// TIA Portal project "Esteira_seletora" (V17)

(* hardware
DEVICE "S7-1500/ET200MP station_1"  S7-1500 station
   slot 0: "Rail_0"  Rack  6ES7 590-1***0-0AA0
   slot 1: "PLC_1"  CPU 1516-3 PN/DP  6ES7 516-3AN02-0AB0  V2.9
      slot 3: "CPU display_1"  6ES7591-1BA00-0AA0
      slot 32768: "PROFINET interface_1"  X1
      slot 33024: "PROFINET interface_2"  X2
      slot 33280: "DP interface_1"  X3
      slot 34817: "Virtual CP interface port_1"  Virtual CP interface port  Virtual CP interface port
   slot 2: "DI 32x24VDC HF_1"  DI 32x24VDC HF  6ES7 521-1BL00-0AB0  V2.2
   slot 3: "DQ 32x24VDC/0.5A HF_1"  DQ 32x24VDC/0.5A HF  6ES7 522-1BL01-0AB0  V1.1
   slot 4: "AI 8xU/I/RTD/TC ST_1"  AI 8xU/I/RTD/TC ST  6ES7 531-7KF00-0AB0  V2.2
   slot 5: "AQ 4xU/I ST_1"  AQ 4xU/I ST  6ES7 532-5HD00-0AB0  V2.2
*)

// ===== PLC "PLC_1"  CPU 1516-3 PN/DP =====

VAR_GLOBAL   // PLC tag table "Default tag table"
   "Liga" AT %I1.1 : Bool;
   "S_capacitivo" AT %I0.0 : Bool;
   "S_indutivo" AT %I0.1 : Bool;
   "S_Peça_peq" AT %I0.4 : Bool;
   "S_Peça_Med" AT %I0.3 : Bool;
   "S_Peça_Grd" AT %I0.2 : Bool;
   "S_Rampa_1" AT %I0.5 : Bool;
   "S_Rampa_2" AT %I0.6 : Bool;
   "S_Rampa_3" AT %I0.7 : Bool;
   "S_Fim_de_Curso" AT %I1.0 : Bool;
   "Motor" AT %Q0.0 : Bool;
   "Cilindro_1" AT %Q0.1 : Bool;
   "Cilindro_2" AT %Q0.2 : Bool;
   "Cilindro_3_Avança" AT %Q0.4 : Bool;
   "Cilindro_3_recuado" AT %Q0.3 : Bool;
   "M_S_capacitivo" AT %M0.0 : Bool;
   "M_S_indutivo" AT %M0.1 : Bool;
   "M_S_Peça_peq" AT %M0.2 : Bool;
   "M_S_Peça_Med" AT %M0.3 : Bool;
   "M_S_Peça_Grd" AT %M0.4 : Bool;
   "Reset" AT %M0.5 : Bool;
   "Count_Rampa_1" AT %MW5 : Int;
   "Count_Rampa_2" AT %MW8 : Int;
   "Count_Rampa_3" AT %MW10 : Int;
   "Count_peca_ok" AT %MW12 : Int;
   "liga_2" AT %M14.0 : Bool;
   "reset_count_2" AT %M14.1 : Bool;
   "reset_manual" AT %I1.2 : Bool;
END_VAR

DATA_BLOCK "Block_1_DB"   // DB1
{ S7_Optimized_Access := 'TRUE' }
VERSION : 0.1
// stored: InstanceOfName Block_1
"Block_1"
BEGIN
END_DATA_BLOCK

// folder: System blocks/Program resources

DATA_BLOCK "rampa1"   // DB2
{ S7_Optimized_Access := 'TRUE' }
AUTHOR : Simatic
FAMILY : IEC
NAME : CNTR
VERSION : 1.0
// stored: InstanceOfName IEC_COUNTER
"IEC_COUNTER"
BEGIN
END_DATA_BLOCK

DATA_BLOCK "rampa2"   // DB3
{ S7_Optimized_Access := 'TRUE' }
AUTHOR : Simatic
FAMILY : IEC
NAME : CNTR
VERSION : 1.0
// stored: InstanceOfName IEC_COUNTER
"IEC_COUNTER"
BEGIN
END_DATA_BLOCK

DATA_BLOCK "rampa3"   // DB4
{ S7_Optimized_Access := 'TRUE' }
AUTHOR : Simatic
FAMILY : IEC
NAME : CNTR
VERSION : 1.0
// stored: InstanceOfName IEC_COUNTER
"IEC_COUNTER"
BEGIN
END_DATA_BLOCK

DATA_BLOCK "peca_OK"   // DB5
{ S7_Optimized_Access := 'TRUE' }
AUTHOR : Simatic
FAMILY : IEC
NAME : CNTR
VERSION : 1.0
// stored: InstanceOfName IEC_COUNTER
"IEC_COUNTER"
BEGIN
END_DATA_BLOCK

// folder: (top level)

FUNCTION_BLOCK "Block_1"   // FB1, GRAPH_PLUS
{ S7_Optimized_Access := 'TRUE' }
VERSION : 0.1
   VAR_INPUT
      OFF_SQ : Bool := false;   // Turn sequence off
      INIT_SQ : Bool := false;   // Set sequence to initial state
      ACK_EF : Bool := false;   // Acknowledge all errors and faults
      S_PREV : Bool := false;   // Output previous step in parameter S_NO
      S_NEXT : Bool := false;   // Indicate next step in parameter S_NO
      SW_AUTO : Bool := false;   // Automatic mode
      SW_TAP : Bool := false;   // Semiautomatic/switch with transition
      SW_TOP : Bool := false;   // Semiautomatic/ignore transition
      SW_MAN : Bool := false;   // Manual mode
      S_SEL : Int := 0;   // Select step to be output to S_NO
      S_ON : Bool := false;   // Activate step indicated in S_NO
      S_OFF : Bool := false;   // Deactivate step indicated S_NO
      T_PUSH : Bool := false;   // Enable transition to switch in semi automatic mode
   END_VAR
   VAR_OUTPUT
      S_NO : Int := 0;   // Step number
      S_MORE : Bool := false;   // More steps are available and can be shown in S_NO
      S_ACTIVE : Bool := false;   // Step indicated in S_NO is active
      ERR_FLT : Bool := false;   // Interlock or supervision group error
      AUTO_ON : Bool := false;   // Automatic mode is active
      TAP_ON : Bool := false;   // Semiautomatic mode/step with transition enabled
      TOP_ON : Bool := false;   // Semiautomatic mode/ignore transition enabled
      MAN_ON : Bool := false;   // Manual mode is active
   END_VAR
   VAR
      HMI_INFO : Array[0..11] of UInt;
      IF_PAR : G7_IfParPlus_V6;
      RT_DATA : G7_RTDataPlus_V6;   // Internal data area
      Trans1 : G7_TransitionPlus_V6;   // Transition structure
      Trans2 : G7_TransitionPlus_V6;   // Transition structure
      Trans3 : G7_TransitionPlus_V6;   // Transition structure
      Trans4 : G7_TransitionPlus_V6;   // Transition structure
      Trans5 : G7_TransitionPlus_V6;   // Transition structure
      Trans6 : G7_TransitionPlus_V6;   // Transition structure
      Trans7 : G7_TransitionPlus_V6;   // Transition structure
      Trans8 : G7_TransitionPlus_V6;   // Transition structure
      Trans9 : G7_TransitionPlus_V6;   // Transition structure
      Trans10 : G7_TransitionPlus_V6;   // Transition structure
      Trans11 : G7_TransitionPlus_V6;   // Transition structure
      stop : G7_StepPlus_V6;   // Step structure
      start : G7_StepPlus_V6;   // Step structure
      pequena : G7_StepPlus_V6;   // Step structure
      grande : G7_StepPlus_V6;   // Step structure
      media : G7_StepPlus_V6;   // Step structure
      Step6 : G7_StepPlus_V6;   // Step structure
      Step7 : G7_StepPlus_V6;   // Step structure
      Step8 : G7_StepPlus_V6;   // Step structure
      platico : G7_StepPlus_V6;   // Step structure
      SINI : Array[0..4] of USInt;
      LSTT : Array[0..10] of USInt;
      ATAJ : Array[0..10] of USInt;
      ATAB : Array[0..10] of USInt;
      PSTT : Array[0..10] of USInt;
      NSTT : Array[0..10] of USInt;
      ASSJ : Array[0..8] of USInt;
      ASSB : Array[0..8] of USInt;
      PTTS : Array[0..8] of USInt;
      NTTS : Array[0..8] of USInt;
      SW_SQTS : Array[0..8] of USInt;
      SWITCH : Array[0..3] of USInt;
      TVX : Array[0..7] of USInt;
      TTX : Array[0..7] of USInt;
      TSX : Array[0..4] of USInt;
      S00X : Array[0..4] of USInt;
      SOFFX : Array[0..4] of USInt;
      SONX : Array[0..4] of USInt;
      SAX : Array[0..4] of USInt;
      SERRX : Array[0..9] of USInt;
      SMX : Array[0..9] of USInt;
      S0X : Array[0..9] of USInt;
      S1X : Array[0..9] of USInt;
      IL_ALARM_INST : Diag_Alarm;
      SUP_ALARM_INST : Diag_Alarm;
      STEP_TIME_ALARM_INST : Diag_Alarm;
      IEC_TIMER_INST : IEC_TIMER;
      TRANSACTION_FLAG : Bool := false;
   END_VAR
   // SINI[0] := 2;
   // SINI[2] := 255;
   // SINI[3] := 255;
   // SINI[4] := 255;
   // LSTT[0] := 255;
   // LSTT[1] := 255;
   // LSTT[2] := 255;
   // LSTT[3] := 255;
   // LSTT[4] := 255;
   // LSTT[5] := 255;
   // LSTT[6] := 1;
   // LSTT[7] := 1;
   // LSTT[8] := 1;
   // LSTT[9] := 1;
   // ATAJ[1] := 1;
   // ATAJ[2] := 2;
   // ATAJ[3] := 3;
   // ATAJ[4] := 4;
   // ATAJ[5] := 5;
   // ATAJ[6] := 6;
   // ATAJ[7] := 7;
   // ATAJ[8] := 8;
   // ATAJ[9] := 9;
   // ATAB[1] := 10;
   // ATAB[2] := 2;
   // ATAB[3] := 1;
   // ATAB[4] := 4;
   // ATAB[5] := 5;
   // ATAB[6] := 6;
   // ATAB[7] := 7;
   // ATAB[8] := 8;
   // ATAB[9] := 9;
   // PSTT[1] := 1;
   // PSTT[2] := 2;
   // PSTT[3] := 1;
   // PSTT[4] := 4;
   // PSTT[5] := 3;
   // PSTT[6] := 5;
   // PSTT[7] := 6;
   // PSTT[8] := 7;
   // PSTT[9] := 8;
   // NSTT[0] := 1;
   // NSTT[1] := 2;
   // NSTT[2] := 5;
   // NSTT[3] := 8;
   // NSTT[4] := 6;
   // NSTT[5] := 7;
   // NSTT[6] := 1;
   // NSTT[7] := 1;
   // NSTT[8] := 1;
   // NSTT[9] := 1;
   // ASSJ[1] := 1;
   // ASSJ[2] := 2;
   // ASSJ[3] := 3;
   // ASSJ[4] := 4;
   // ASSJ[5] := 5;
   // ASSJ[6] := 6;
   // ASSJ[7] := 7;
   // ASSJ[8] := 8;
   // ASSB[1] := 1;
   // ASSB[2] := 4;
   // ASSB[3] := 2;
   // ASSB[4] := 3;
   // ASSB[5] := 5;
   // ASSB[6] := 6;
   // ASSB[7] := 7;
   // ASSB[8] := 8;
   // PTTS[0] := 255;
   // PTTS[2] := 1;
   // PTTS[3] := 1;
   // PTTS[4] := 1;
   // PTTS[5] := 2;
   // PTTS[6] := 4;
   // PTTS[7] := 5;
   // PTTS[8] := 3;
   // NTTS[1] := 1;
   // NTTS[2] := 2;
   // NTTS[3] := 5;
   // NTTS[4] := 4;
   // NTTS[5] := 6;
   // NTTS[6] := 7;
   // NTTS[7] := 8;
   // NTTS[8] := 9;
   // SW_SQTS[2] := 1;
   // SW_SQTS[3] := 2;
   // SW_SQTS[4] := 3;
   // SW_SQTS[5] := 1;
   // SW_SQTS[6] := 3;
   // SW_SQTS[7] := 2;
   // SW_SQTS[8] := 4;
   // SWITCH[0] := 128;
   // SWITCH[1] := 41;
   // SWITCH[2] := 3;
   // TVX[0] := 16#1;
   // TTX[0] := 16#1;
   // TSX[0] := 16#1;
   // S00X[0] := 16#1;
   // SOFFX[0] := 16#1;
   // SONX[0] := 16#1;
   // SAX[0] := 16#1;
   // SERRX[0] := 16#1;
   // SMX[0] := 16#1;
   // S0X[0] := 16#1;
   // S1X[0] := 16#1;
   // ATAJ[10] := 10;
   // ATAB[10] := 3;
   // PSTT[10] := 1;
BEGIN
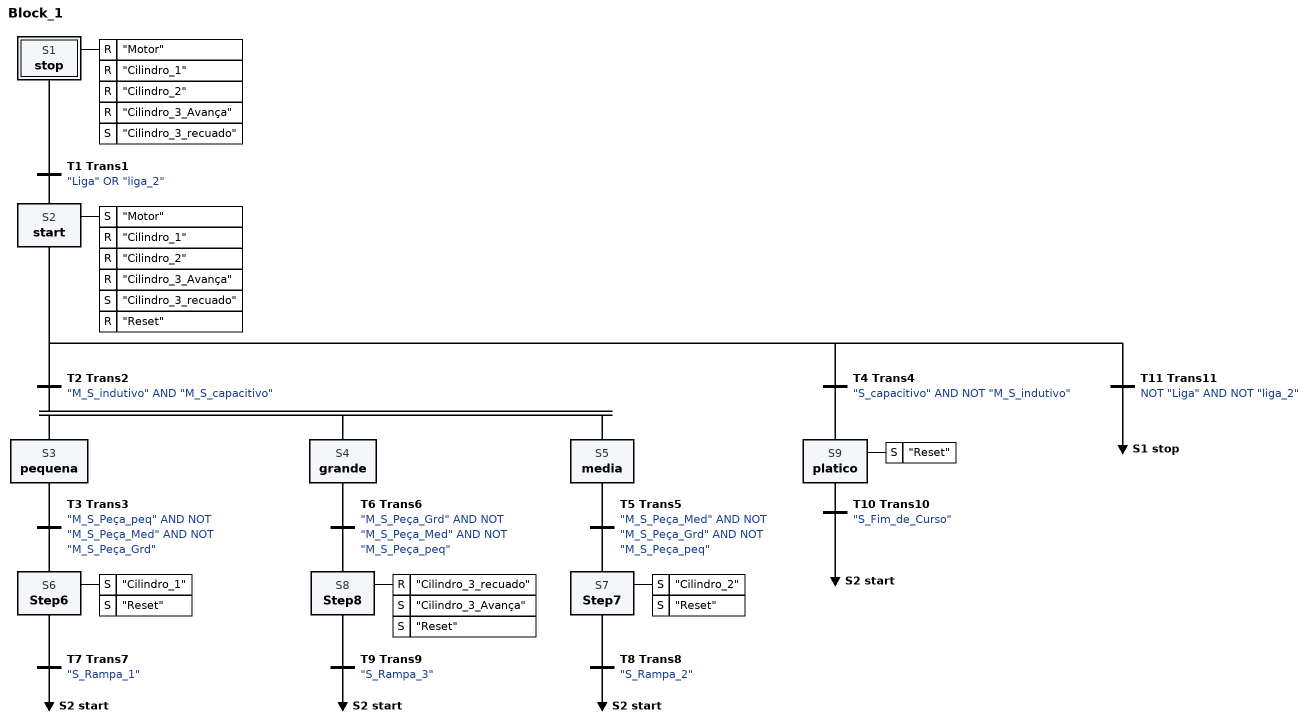
   // sequencer 1
   INITIAL_STEP stop:   // S1, max time T#10S, warning time T#7S
              R    "Motor"
              R    "Cilindro_1"
              R    "Cilindro_2"
              R    "Cilindro_3_Avança"
              S    "Cilindro_3_recuado"
   END_STEP
   TRANSITION Trans1 FROM stop TO start   // T1
      := "Liga" OR "liga_2";
   END_TRANSITION
   STEP start:   // S2, max time T#10S, warning time T#7S
              S    "Motor"
              R    "Cilindro_1"
              R    "Cilindro_2"
              R    "Cilindro_3_Avança"
              S    "Cilindro_3_recuado"
              R    "Reset"
   END_STEP
   TRANSITION Trans2 FROM start TO (pequena, grande, media)   // T2
      := "M_S_indutivo" AND "M_S_capacitivo";
   END_TRANSITION
   TRANSITION Trans4 FROM start TO platico   // T4
      := "S_capacitivo" AND NOT "M_S_indutivo";
   END_TRANSITION
   TRANSITION Trans11 FROM start TO stop   // T11, jump
      := NOT "Liga" AND NOT "liga_2";
   END_TRANSITION
   STEP pequena:   // S3, max time T#10S, warning time T#7S
   END_STEP
   TRANSITION Trans3 FROM pequena TO Step6   // T3
      := "M_S_Peça_peq" AND NOT "M_S_Peça_Med" AND NOT "M_S_Peça_Grd";
   END_TRANSITION
   STEP grande:   // S4, max time T#10S, warning time T#7S
   END_STEP
   TRANSITION Trans6 FROM grande TO Step8   // T6
      := "M_S_Peça_Grd" AND NOT "M_S_Peça_Med" AND NOT "M_S_Peça_peq";
   END_TRANSITION
   STEP media:   // S5, max time T#10S, warning time T#7S
   END_STEP
   TRANSITION Trans5 FROM media TO Step7   // T5
      := "M_S_Peça_Med" AND NOT "M_S_Peça_Grd" AND NOT "M_S_Peça_peq";
   END_TRANSITION
   STEP Step6:   // S6, max time T#10S, warning time T#7S
              S    "Cilindro_1"
              S    "Reset"
   END_STEP
   TRANSITION Trans7 FROM Step6 TO start   // T7, jump
      := "S_Rampa_1";
   END_TRANSITION
   STEP Step7:   // S7, max time T#10S, warning time T#7S
              S    "Cilindro_2"
              S    "Reset"
   END_STEP
   TRANSITION Trans8 FROM Step7 TO start   // T8, jump
      := "S_Rampa_2";
   END_TRANSITION
   STEP Step8:   // S8, max time T#10S, warning time T#7S
              R    "Cilindro_3_recuado"
              S    "Cilindro_3_Avança"
              S    "Reset"
   END_STEP
   TRANSITION Trans9 FROM Step8 TO start   // T9, jump
      := "S_Rampa_3";
   END_TRANSITION
   STEP platico:   // S9, max time T#10S, warning time T#7S
              S    "Reset"
   END_STEP
   TRANSITION Trans10 FROM platico TO start   // T10, jump
      := "S_Fim_de_Curso";
   END_TRANSITION
END_FUNCTION_BLOCK

FUNCTION "Block_2" : Void   // FC1, LAD
{ S7_Optimized_Access := 'TRUE' }
VERSION : 0.1
BEGIN

REGION Network 1
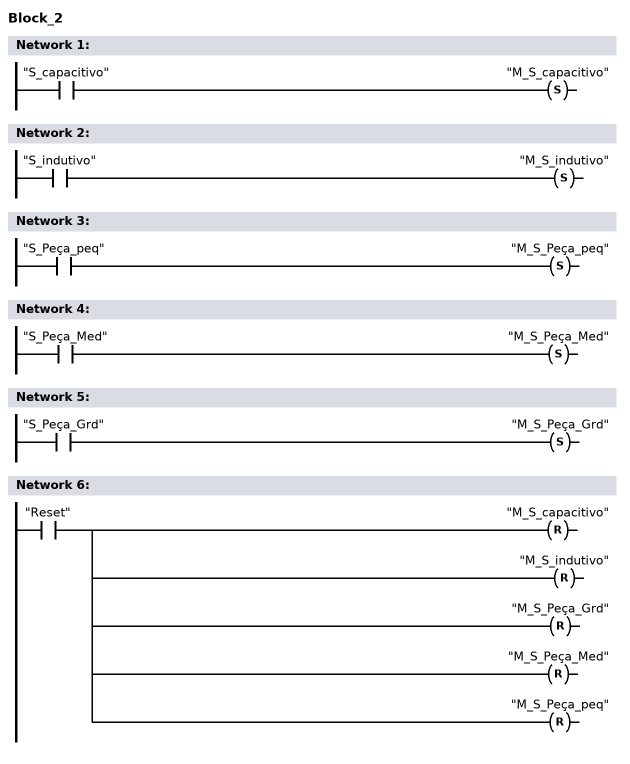
   RUNG wire#powerrail
      Contact( "S_capacitivo" )
      S_Coil( "M_S_capacitivo" )
   END_RUNG
   // the same network as SCL:
   IF "S_capacitivo" THEN "M_S_capacitivo" := TRUE; END_IF;
END_REGION

REGION Network 2
   RUNG wire#powerrail
      Contact( "S_indutivo" )
      S_Coil( "M_S_indutivo" )
   END_RUNG
   // the same network as SCL:
   IF "S_indutivo" THEN "M_S_indutivo" := TRUE; END_IF;
END_REGION

REGION Network 3
   RUNG wire#powerrail
      Contact( "S_Peça_peq" )
      S_Coil( "M_S_Peça_peq" )
   END_RUNG
   // the same network as SCL:
   IF "S_Peça_peq" THEN "M_S_Peça_peq" := TRUE; END_IF;
END_REGION

REGION Network 4
   RUNG wire#powerrail
      Contact( "S_Peça_Med" )
      S_Coil( "M_S_Peça_Med" )
   END_RUNG
   // the same network as SCL:
   IF "S_Peça_Med" THEN "M_S_Peça_Med" := TRUE; END_IF;
END_REGION

REGION Network 5
   RUNG wire#powerrail
      Contact( "S_Peça_Grd" )
      S_Coil( "M_S_Peça_Grd" )
   END_RUNG
   // the same network as SCL:
   IF "S_Peça_Grd" THEN "M_S_Peça_Grd" := TRUE; END_IF;
END_REGION

REGION Network 6
   RUNG wire#powerrail
      Contact( "Reset" )
      wire#w1
      R_Coil( "M_S_capacitivo" )
   END_RUNG
   RUNG wire#w1
      R_Coil( "M_S_indutivo" )
   END_RUNG
   RUNG wire#w1
      R_Coil( "M_S_Peça_Grd" )
   END_RUNG
   RUNG wire#w1
      R_Coil( "M_S_Peça_Med" )
   END_RUNG
   RUNG wire#w1
      R_Coil( "M_S_Peça_peq" )
   END_RUNG
   // the same network as SCL:
   IF "Reset" THEN
       "M_S_capacitivo" := FALSE;
       "M_S_indutivo" := FALSE;
       "M_S_Peça_Grd" := FALSE;
       "M_S_Peça_Med" := FALSE;
       "M_S_Peça_peq" := FALSE;
   END_IF;
END_REGION
END_FUNCTION

ORGANIZATION_BLOCK "Main"   // OB1, LAD, ProgramCycle
TITLE = "Main Program Sweep (Cycle)"
{ S7_Optimized_Access := 'TRUE' }
VERSION : 0.1
   VAR_INPUT
      Initial_Call : Bool;   // Initial call of this OB
      Remanence : Bool;   // =True, if remanent data are available
   END_VAR
BEGIN

REGION Network 1
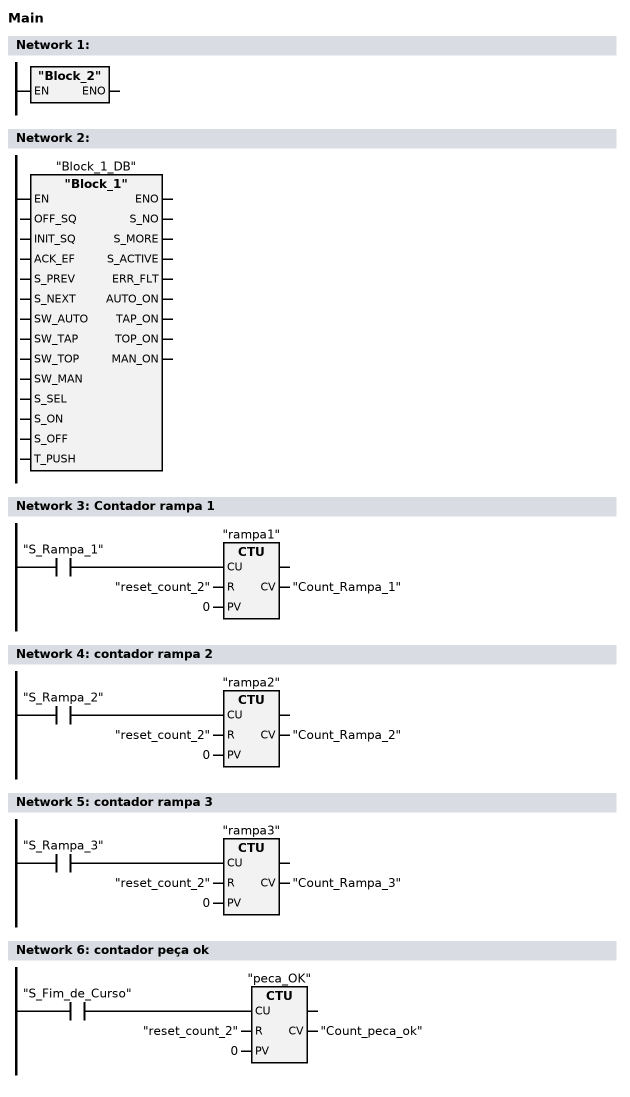
   RUNG wire#powerrail
      "Block_2"()
   END_RUNG
   // the same network as SCL:
   "Block_2"();
END_REGION

REGION Network 2
   RUNG wire#powerrail
      "Block_1_DB"(OFF_SQ :=, INIT_SQ :=, ACK_EF :=, S_PREV :=, S_NEXT :=, SW_AUTO :=, SW_TAP :=, SW_TOP :=, SW_MAN :=, S_SEL :=, S_ON :=, S_OFF :=, T_PUSH :=, S_NO =>, S_MORE =>, S_ACTIVE =>, ERR_FLT =>, AUTO_ON =>, TAP_ON =>, TOP_ON =>, MAN_ON =>)
   END_RUNG
   // the same network as SCL:
   "Block_1_DB"();   // "Block_1"
END_REGION

REGION Network 3: Contador rampa 1
   "rampa1".CTU(CU := "S_Rampa_1", R := "reset_count_2", PV := 0, CV => "Count_Rampa_1");
END_REGION

REGION Network 4: contador rampa 2
   "rampa2".CTU(CU := "S_Rampa_2", R := "reset_count_2", PV := 0, CV => "Count_Rampa_2");
END_REGION

REGION Network 5: contador rampa 3
   "rampa3".CTU(CU := "S_Rampa_3", R := "reset_count_2", PV := 0, CV => "Count_Rampa_3");
END_REGION

REGION Network 6: contador peça ok
   "peca_OK".CTU(CU := "S_Fim_de_Curso", R := "reset_count_2", PV := 0, CV => "Count_peca_ok");
END_REGION
END_ORGANIZATION_BLOCK